PROGRAM MAIN
VAR
	
END_VAR

END_PROGRAM

(* stored: Version 1.1.0.1, ProductVersion 3.1.4024.12
   POU MAIN: Id {f9c32a99-8e78-4f74-88a7-234889507b85}, SpecialFunc None *)
